FUNCTION_BLOCK ButtonDs (* Basic Function Block Type *)
  (* Standard: 61499-2 *)
  (* Version 0.0, 12/23/2020, midhu, nxtControl GmbH, Template *)
  PACKAGE Main;
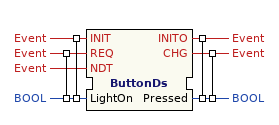
  EVENT_INPUT
    INIT WITH LightOn;
    REQ WITH LightOn; (* Initialization Request *)
    NDT; (* Non deterministic transition *)
  END_EVENT
  EVENT_OUTPUT
    INITO WITH Pressed;
    CHG WITH Pressed; (* Initialization Confirm *)
  END_EVENT
  VAR_INPUT
    LightOn : BOOL; (* Input event qualifier *)
  END_VAR
  VAR_OUTPUT
    Pressed : BOOL; (* Output event qualifier *)
  END_VAR
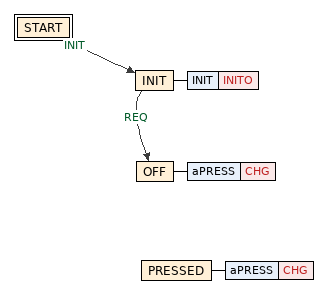
  EC_STATES
    START; (* Initial State *)
    INIT : INIT -> INITO; (* Initialization *)
    OFF : aPRESS -> CHG;
    PRESSED : aPRESS -> CHG;
  END_STATES
  EC_TRANSITIONS
    START TO INIT := INIT;
    INIT TO OFF := REQ;
  END_TRANSITIONS
  ALGORITHM INIT IN ST: (* Initialization algorithm *)
Pressed:=FALSE;
  END_ALGORITHM
  ALGORITHM aOFF IN ST:
Pressed:=FALSE;
  END_ALGORITHM
  ALGORITHM aPRESS IN ST:
Pressed:=TRUE;
  END_ALGORITHM
END_FUNCTION_BLOCK
